{attribute 'reflection'} 
FUNCTION_BLOCK FB_instancePath 
VAR 
    {attribute 'instance-path'} 
    {attribute 'noinit'} 
    sPath : STRING; 
END_VAR

END_FUNCTION_BLOCK

(* stored: Version 1.1.0.1, ProductVersion 3.1.4022.16
   POU FB_instancePath: Id {819d84ae-5755-4f81-b04d-000bd20f24c0}, SpecialFunc None *)
